// TIA Portal project "BTL2_TIA" (V17)

(* hardware
DEVICE "S7-300/ET200M station_2"  S7-300 station
   slot 0: "Rail_0"  Rail  6ES7 390-1***0-0AA0
   slot 2: "PLC_2"  CPU 314C-2 PN/DP  6ES7 314-6EH04-0AB0  V3.3
      slot 2: "PROFINET interface_1"  PN-IO
         slot 1: "Port_1"  Port
         slot 2: "Port_2"  Port
      slot 5: "DI 24/DO 16_1"  DI24/DO16
      slot 6: "AI 5/AO 2_1"  AI5/AO2
      slot 7: "Count_1"  Counter
      slot 8: "Positioning_1"  Positioning
*)

// ===== PLC "PLC_2"  CPU 314C-2 PN/DP =====

VAR_GLOBAL   // PLC tag table "I"
   "Start" AT %I0.0 : Bool;
   "Stop" AT %I0.1 : Bool;
   "Reset" AT %I0.2 : Bool;
   "Emer" AT %I0.3 : Bool;
   "Mode" AT %I0.4 : Bool;
   "S1" AT %I1.0 : Bool;   // A1
   "S2" AT %I1.1 : Bool;   // A0
   "S3" AT %I1.2 : Bool;   // B1
   "S4" AT %I1.3 : Bool;   // B0
   "S5" AT %I1.4 : Bool;   // C1
   "S6" AT %I1.5 : Bool;   // C0
   "cell" AT %I0.5 : Bool;
   "swa+" AT %I2.0 : Bool;
   "swa-" AT %I2.1 : Bool;
   "swb+" AT %I2.2 : Bool;
   "swb-" AT %I2.3 : Bool;
   "swc+" AT %I2.4 : Bool;
   "swc-" AT %I2.5 : Bool;
   "sm" AT %I2.6 : Bool;
END_VAR

VAR_GLOBAL   // PLC tag table "M"
   "k1-au" AT %M0.1 : Bool;
   "k2-au" AT %M0.2 : Bool;
   "k3-au" AT %M0.3 : Bool;
   "k4-au" AT %M0.4 : Bool;
   "k5-au" AT %M0.5 : Bool;
   "k6-au" AT %M0.6 : Bool;
   "k7-au" AT %M0.7 : Bool;
   "k0-au" AT %M0.0 : Bool;
   "cell_temp" AT %M1.0 : Bool;
   "LED_1hz" AT %M1.1 : Bool;
   "LED_Stable" AT %M1.2 : Bool;
   "au-manu" AT %M1.3 : Bool;
   "manu-au" AT %M1.4 : Bool;
   "k0-manu" AT %M1.5 : Bool;
   "protocol" AT %M1.7 : Bool;
   "k0_manu1" AT %M2.0 : Bool;
   "cell_temp_manual" AT %M2.1 : Bool;
   "stop temporary" AT %M2.2 : Bool;
   "m_err1" AT %M10.1 : Bool;
   "m_err2" AT %M10.2 : Bool;
   "m_err3" AT %M10.3 : Bool;
   "tag 1 auto" AT %M20.1 : Bool;
   "tag 2 auto" AT %M20.2 : Bool;
   "tag 1 manual" AT %M20.3 : Bool;
   "tag 2 manual" AT %M20.4 : Bool;
   "state 1" AT %M20.5 : Bool;
   "state 2" AT %M20.6 : Bool;
   "state 3" AT %M20.7 : Bool;
   "tag1" AT %M21.0 : Bool;
END_VAR

VAR_GLOBAL   // PLC tag table "Q"
   "Y1" AT %Q0.0 : Bool;   // A+
   "Y2" AT %Q0.1 : Bool;   // A-
   "Y3" AT %Q0.2 : Bool;   // B+
   "Y4" AT %Q0.3 : Bool;   // B-
   "Y5" AT %Q0.4 : Bool;   // C+
   "Y6" AT %Q0.5 : Bool;   // C-
   "M" AT %Q1.0 : Bool;
   "cell LED" AT %Q1.1 : Bool;
   "auto LED" AT %Q1.2 : Bool;
   "manual LED" AT %Q1.3 : Bool;
   "ready LED" AT %Q1.4 : Bool;
   "err1" AT %Q1.5 : Bool;
   "err2" AT %Q1.6 : Bool;
   "err3" AT %Q1.7 : Bool;
END_VAR

FUNCTION "auto" : Void   // FC1, LAD
{ S7_Optimized_Access := 'FALSE' }
VERSION : 0.1
BEGIN

REGION Network 1
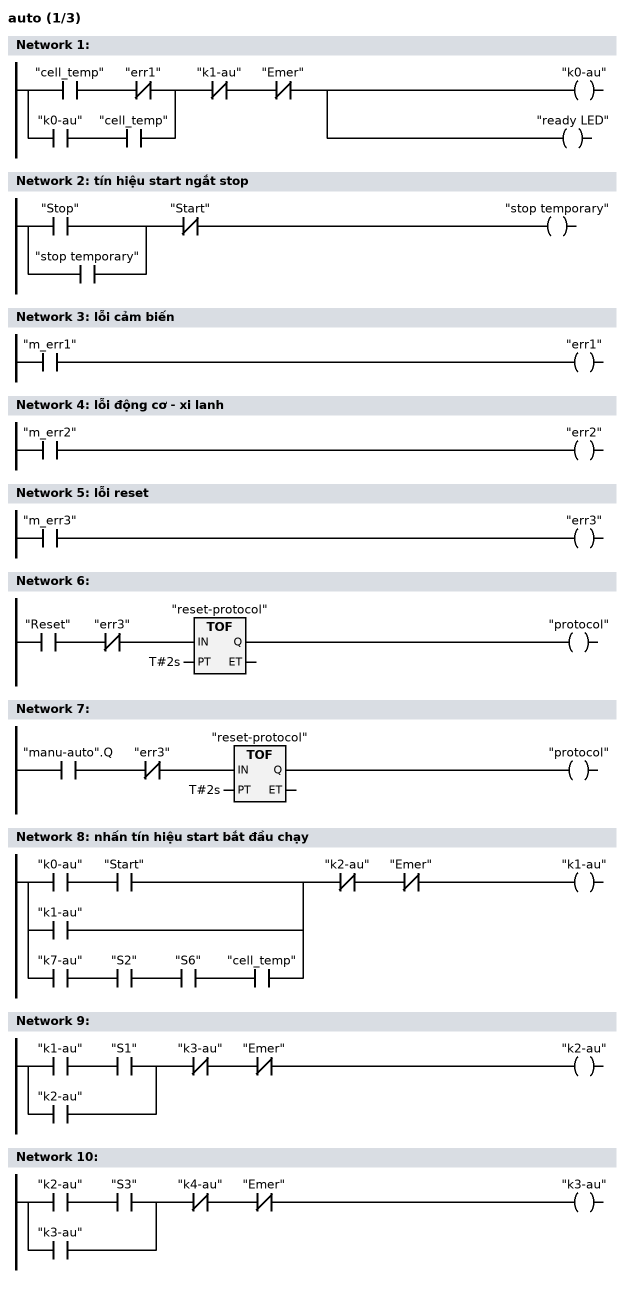
   RUNG wire#powerrail
      Contact( "cell_temp" )
      I_Contact( "err1" )
      wire#w1
      I_Contact( "k1-au" )
      I_Contact( "Emer" )
      wire#w2
      Coil( "k0-au" )
   END_RUNG
   RUNG wire#powerrail
      Contact( "k0-au" )
      Contact( "cell_temp" )
   END_RUNG wire#w1
   RUNG wire#w2
      Coil( "ready LED" )
   END_RUNG
   // the same network as SCL:
   "k0-au" := (("cell_temp" AND NOT "err1") OR ("k0-au" AND "cell_temp")) AND NOT "k1-au" AND NOT "Emer";
   "ready LED" := "k0-au";
END_REGION

REGION Network 2: tín hiệu start ngắt stop
   RUNG wire#powerrail
      Contact( "Stop" )
      wire#w1
      I_Contact( "Start" )
      Coil( "stop temporary" )
   END_RUNG
   RUNG wire#powerrail
      Contact( "stop temporary" )
   END_RUNG wire#w1
   // the same network as SCL:
   "stop temporary" := ("Stop" OR "stop temporary") AND NOT "Start";
END_REGION

REGION Network 3: lỗi cảm biến
   RUNG wire#powerrail
      Contact( "m_err1" )
      Coil( "err1" )
   END_RUNG
   // the same network as SCL:
   "err1" := "m_err1";
END_REGION

REGION Network 4: lỗi động cơ - xi lanh
   RUNG wire#powerrail
      Contact( "m_err2" )
      Coil( "err2" )
   END_RUNG
   // the same network as SCL:
   "err2" := "m_err2";
END_REGION

REGION Network 5: lỗi reset
   RUNG wire#powerrail
      Contact( "m_err3" )
      Coil( "err3" )
   END_RUNG
   // the same network as SCL:
   "err3" := "m_err3";
END_REGION

REGION Network 6
   "reset-protocol".TOF(IN := "Reset" AND NOT "err3", PT := T#2s);
   "protocol" := "reset-protocol".Q;
END_REGION

REGION Network 7
   "reset-protocol".TOF(IN := "manu-auto".Q AND NOT "err3", PT := T#2s);
   "protocol" := "reset-protocol".Q;
END_REGION

REGION Network 8: nhấn tín hiệu start bắt đầu chạy
   RUNG wire#powerrail
      Contact( "k0-au" )
      Contact( "Start" )
      wire#w1
      I_Contact( "k2-au" )
      I_Contact( "Emer" )
      Coil( "k1-au" )
   END_RUNG
   RUNG wire#powerrail
      Contact( "k1-au" )
   END_RUNG wire#w1
   RUNG wire#powerrail
      Contact( "k7-au" )
      Contact( "S2" )
      Contact( "S6" )
      Contact( "cell_temp" )
   END_RUNG wire#w1
   // the same network as SCL:
   "k1-au" := (("k0-au" AND "Start") OR "k1-au" OR ("k7-au" AND "S2" AND "S6" AND "cell_temp")) AND NOT "k2-au" AND NOT "Emer";
END_REGION

REGION Network 9
   RUNG wire#powerrail
      Contact( "k1-au" )
      Contact( "S1" )
      wire#w1
      I_Contact( "k3-au" )
      I_Contact( "Emer" )
      Coil( "k2-au" )
   END_RUNG
   RUNG wire#powerrail
      Contact( "k2-au" )
   END_RUNG wire#w1
   // the same network as SCL:
   "k2-au" := (("k1-au" AND "S1") OR "k2-au") AND NOT "k3-au" AND NOT "Emer";
END_REGION

REGION Network 10
   RUNG wire#powerrail
      Contact( "k2-au" )
      Contact( "S3" )
      wire#w1
      I_Contact( "k4-au" )
      I_Contact( "Emer" )
      Coil( "k3-au" )
   END_RUNG
   RUNG wire#powerrail
      Contact( "k3-au" )
   END_RUNG wire#w1
   // the same network as SCL:
   "k3-au" := (("k2-au" AND "S3") OR "k3-au") AND NOT "k4-au" AND NOT "Emer";
END_REGION

REGION Network 11
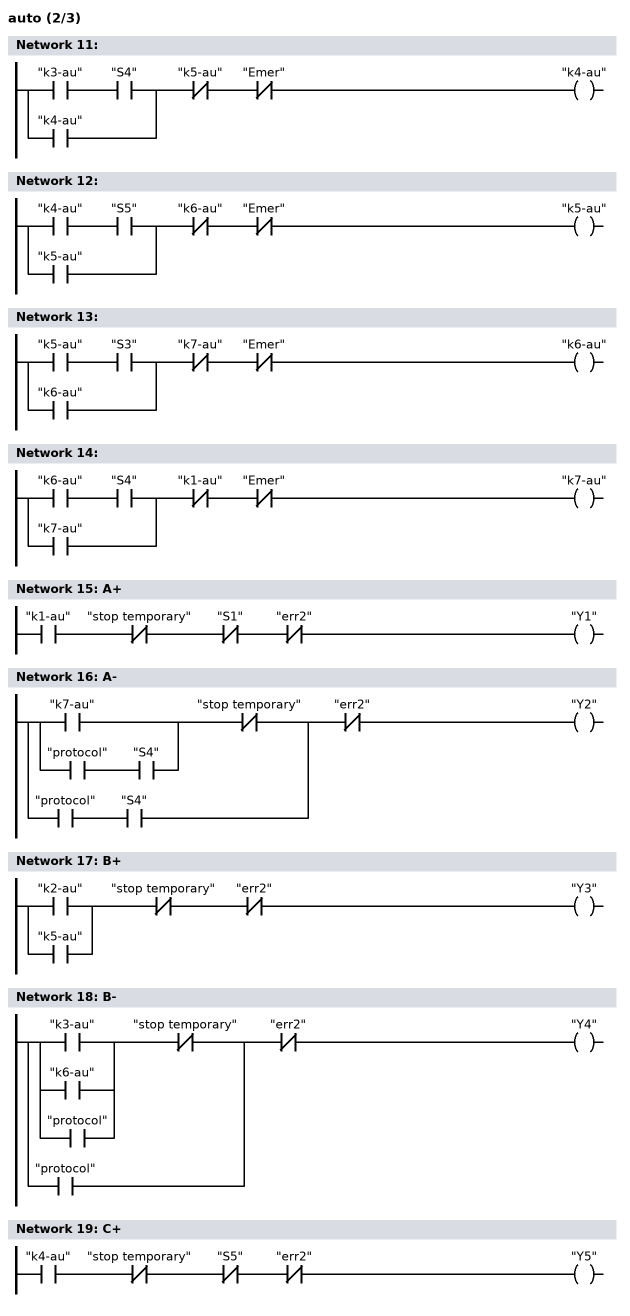
   RUNG wire#powerrail
      Contact( "k3-au" )
      Contact( "S4" )
      wire#w1
      I_Contact( "k5-au" )
      I_Contact( "Emer" )
      Coil( "k4-au" )
   END_RUNG
   RUNG wire#powerrail
      Contact( "k4-au" )
   END_RUNG wire#w1
   // the same network as SCL:
   "k4-au" := (("k3-au" AND "S4") OR "k4-au") AND NOT "k5-au" AND NOT "Emer";
END_REGION

REGION Network 12
   RUNG wire#powerrail
      Contact( "k4-au" )
      Contact( "S5" )
      wire#w1
      I_Contact( "k6-au" )
      I_Contact( "Emer" )
      Coil( "k5-au" )
   END_RUNG
   RUNG wire#powerrail
      Contact( "k5-au" )
   END_RUNG wire#w1
   // the same network as SCL:
   "k5-au" := (("k4-au" AND "S5") OR "k5-au") AND NOT "k6-au" AND NOT "Emer";
END_REGION

REGION Network 13
   RUNG wire#powerrail
      Contact( "k5-au" )
      Contact( "S3" )
      wire#w1
      I_Contact( "k7-au" )
      I_Contact( "Emer" )
      Coil( "k6-au" )
   END_RUNG
   RUNG wire#powerrail
      Contact( "k6-au" )
   END_RUNG wire#w1
   // the same network as SCL:
   "k6-au" := (("k5-au" AND "S3") OR "k6-au") AND NOT "k7-au" AND NOT "Emer";
END_REGION

REGION Network 14
   RUNG wire#powerrail
      Contact( "k6-au" )
      Contact( "S4" )
      wire#w1
      I_Contact( "k1-au" )
      I_Contact( "Emer" )
      Coil( "k7-au" )
   END_RUNG
   RUNG wire#powerrail
      Contact( "k7-au" )
   END_RUNG wire#w1
   // the same network as SCL:
   "k7-au" := (("k6-au" AND "S4") OR "k7-au") AND NOT "k1-au" AND NOT "Emer";
END_REGION

REGION Network 15: A+
   RUNG wire#powerrail
      Contact( "k1-au" )
      I_Contact( "stop temporary" )
      I_Contact( "S1" )
      I_Contact( "err2" )
      Coil( "Y1" )
   END_RUNG
   // the same network as SCL:
   "Y1" := "k1-au" AND NOT "stop temporary" AND NOT "S1" AND NOT "err2";
END_REGION

REGION Network 16: A-
   RUNG wire#powerrail
      Contact( "k7-au" )
      wire#w1
      I_Contact( "stop temporary" )
      wire#w2
      I_Contact( "err2" )
      Coil( "Y2" )
   END_RUNG
   RUNG wire#powerrail
      Contact( "protocol" )
      Contact( "S4" )
   END_RUNG wire#w1
   RUNG wire#powerrail
      Contact( "protocol" )
      Contact( "S4" )
   END_RUNG wire#w2
   // the same network as SCL:
   "Y2" := ((("k7-au" OR ("protocol" AND "S4")) AND NOT "stop temporary") OR ("protocol" AND "S4")) AND NOT "err2";
END_REGION

REGION Network 17: B+
   RUNG wire#powerrail
      Contact( "k2-au" )
      wire#w1
      I_Contact( "stop temporary" )
      I_Contact( "err2" )
      Coil( "Y3" )
   END_RUNG
   RUNG wire#powerrail
      Contact( "k5-au" )
   END_RUNG wire#w1
   // the same network as SCL:
   "Y3" := ("k2-au" OR "k5-au") AND NOT "stop temporary" AND NOT "err2";
END_REGION

REGION Network 18: B-
   RUNG wire#powerrail
      Contact( "k3-au" )
      wire#w1
      I_Contact( "stop temporary" )
      wire#w2
      I_Contact( "err2" )
      Coil( "Y4" )
   END_RUNG
   RUNG wire#powerrail
      Contact( "k6-au" )
   END_RUNG wire#w1
   RUNG wire#powerrail
      Contact( "protocol" )
   END_RUNG wire#w1
   RUNG wire#powerrail
      Contact( "protocol" )
   END_RUNG wire#w2
   // the same network as SCL:
   "Y4" := ((("k3-au" OR "k6-au" OR "protocol") AND NOT "stop temporary") OR "protocol") AND NOT "err2";
END_REGION

REGION Network 19: C+
   RUNG wire#powerrail
      Contact( "k4-au" )
      I_Contact( "stop temporary" )
      I_Contact( "S5" )
      I_Contact( "err2" )
      Coil( "Y5" )
   END_RUNG
   // the same network as SCL:
   "Y5" := "k4-au" AND NOT "stop temporary" AND NOT "S5" AND NOT "err2";
END_REGION

REGION Network 20: C-
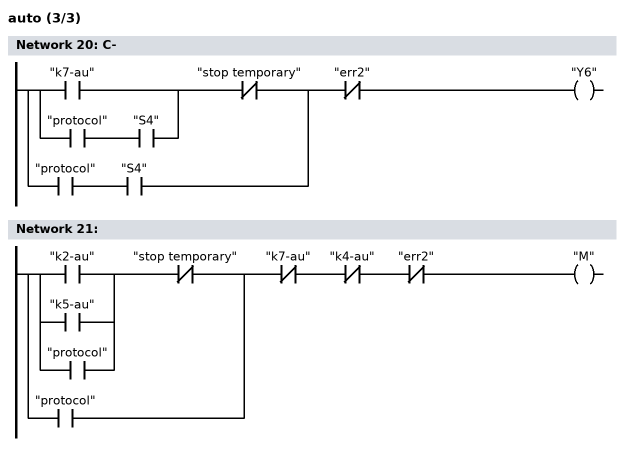
   RUNG wire#powerrail
      Contact( "k7-au" )
      wire#w1
      I_Contact( "stop temporary" )
      wire#w2
      I_Contact( "err2" )
      Coil( "Y6" )
   END_RUNG
   RUNG wire#powerrail
      Contact( "protocol" )
      Contact( "S4" )
   END_RUNG wire#w1
   RUNG wire#powerrail
      Contact( "protocol" )
      Contact( "S4" )
   END_RUNG wire#w2
   // the same network as SCL:
   "Y6" := ((("k7-au" OR ("protocol" AND "S4")) AND NOT "stop temporary") OR ("protocol" AND "S4")) AND NOT "err2";
END_REGION

REGION Network 21
   RUNG wire#powerrail
      Contact( "k2-au" )
      wire#w1
      I_Contact( "stop temporary" )
      wire#w2
      I_Contact( "k7-au" )
      I_Contact( "k4-au" )
      I_Contact( "err2" )
      Coil( "M" )
   END_RUNG
   RUNG wire#powerrail
      Contact( "k5-au" )
   END_RUNG wire#w1
   RUNG wire#powerrail
      Contact( "protocol" )
   END_RUNG wire#w1
   RUNG wire#powerrail
      Contact( "protocol" )
   END_RUNG wire#w2
   // the same network as SCL:
   "M" := ((("k2-au" OR "k5-au" OR "protocol") AND NOT "stop temporary") OR "protocol") AND NOT "k7-au" AND NOT "k4-au" AND NOT "err2";
END_REGION
END_FUNCTION

FUNCTION "manu" : Void   // FC2, LAD
{ S7_Optimized_Access := 'FALSE' }
VERSION : 0.1
   VAR_TEMP   // added for the SCL form of the ladder/FBD networks
      _w1 : Bool;
      _w2 : Bool;
   END_VAR
BEGIN

REGION Network 1: reset-from-auto
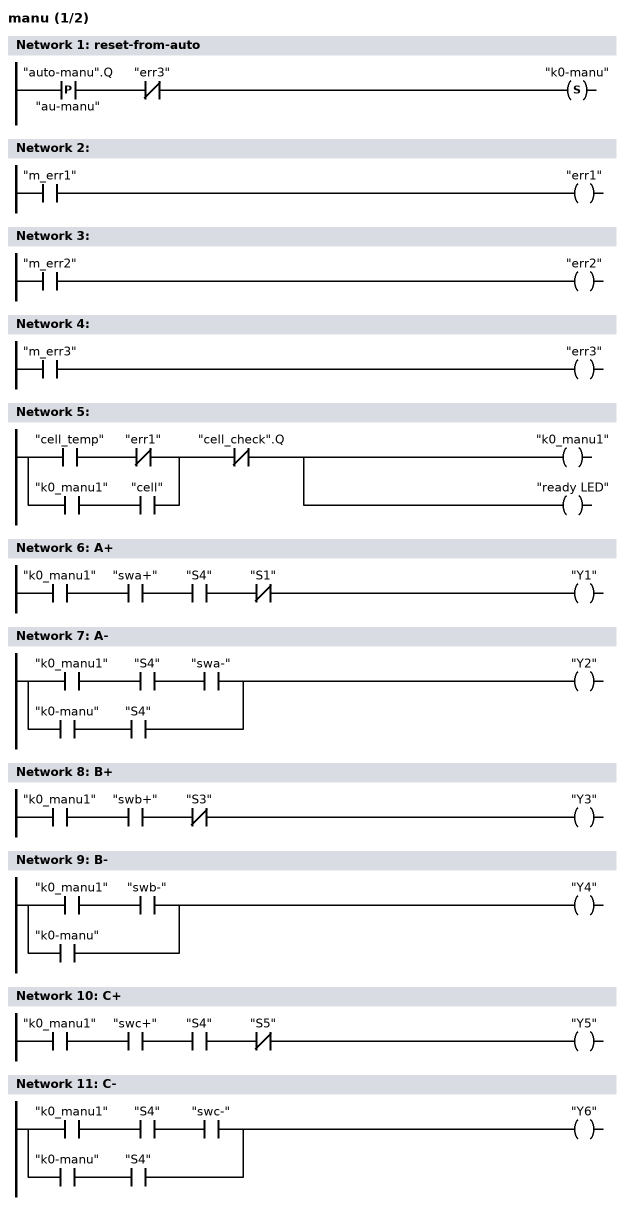
   RUNG wire#powerrail
      P_Contact(operand := "auto-manu".Q, bit := "au-manu")
      I_Contact( "err3" )
      S_Coil( "k0-manu" )
   END_RUNG
   // the same network as SCL:
   #_w1 := "auto-manu".Q AND NOT "au-manu";   // rising edge of "auto-manu".Q
   "au-manu" := "auto-manu".Q;
   IF #_w1 AND NOT "err3" THEN "k0-manu" := TRUE; END_IF;
END_REGION

REGION Network 2
   RUNG wire#powerrail
      Contact( "m_err1" )
      Coil( "err1" )
   END_RUNG
   // the same network as SCL:
   "err1" := "m_err1";
END_REGION

REGION Network 3
   RUNG wire#powerrail
      Contact( "m_err2" )
      Coil( "err2" )
   END_RUNG
   // the same network as SCL:
   "err2" := "m_err2";
END_REGION

REGION Network 4
   RUNG wire#powerrail
      Contact( "m_err3" )
      Coil( "err3" )
   END_RUNG
   // the same network as SCL:
   "err3" := "m_err3";
END_REGION

REGION Network 5
   RUNG wire#powerrail
      Contact( "cell_temp" )
      I_Contact( "err1" )
      wire#w1
      I_Contact( "cell_check".Q )
      wire#w2
      Coil( "k0_manu1" )
   END_RUNG
   RUNG wire#powerrail
      Contact( "k0_manu1" )
      Contact( "cell" )
   END_RUNG wire#w1
   RUNG wire#w2
      Coil( "ready LED" )
   END_RUNG
   // the same network as SCL:
   "k0_manu1" := (("cell_temp" AND NOT "err1") OR ("k0_manu1" AND "cell")) AND NOT "cell_check".Q;
   "ready LED" := "k0_manu1";
END_REGION

REGION Network 6: A+
   RUNG wire#powerrail
      Contact( "k0_manu1" )
      Contact( "swa+" )
      Contact( "S4" )
      I_Contact( "S1" )
      Coil( "Y1" )
   END_RUNG
   // the same network as SCL:
   "Y1" := "k0_manu1" AND "swa+" AND "S4" AND NOT "S1";
END_REGION

REGION Network 7: A-
   RUNG wire#powerrail
      Contact( "k0_manu1" )
      Contact( "S4" )
      Contact( "swa-" )
      wire#w1
      Coil( "Y2" )
   END_RUNG
   RUNG wire#powerrail
      Contact( "k0-manu" )
      Contact( "S4" )
   END_RUNG wire#w1
   // the same network as SCL:
   "Y2" := ("k0_manu1" AND "S4" AND "swa-") OR ("k0-manu" AND "S4");
END_REGION

REGION Network 8: B+
   RUNG wire#powerrail
      Contact( "k0_manu1" )
      Contact( "swb+" )
      I_Contact( "S3" )
      Coil( "Y3" )
   END_RUNG
   // the same network as SCL:
   "Y3" := "k0_manu1" AND "swb+" AND NOT "S3";
END_REGION

REGION Network 9: B-
   RUNG wire#powerrail
      Contact( "k0_manu1" )
      Contact( "swb-" )
      wire#w1
      Coil( "Y4" )
   END_RUNG
   RUNG wire#powerrail
      Contact( "k0-manu" )
   END_RUNG wire#w1
   // the same network as SCL:
   "Y4" := ("k0_manu1" AND "swb-") OR "k0-manu";
END_REGION

REGION Network 10: C+
   RUNG wire#powerrail
      Contact( "k0_manu1" )
      Contact( "swc+" )
      Contact( "S4" )
      I_Contact( "S5" )
      Coil( "Y5" )
   END_RUNG
   // the same network as SCL:
   "Y5" := "k0_manu1" AND "swc+" AND "S4" AND NOT "S5";
END_REGION

REGION Network 11: C-
   RUNG wire#powerrail
      Contact( "k0_manu1" )
      Contact( "S4" )
      Contact( "swc-" )
      wire#w1
      Coil( "Y6" )
   END_RUNG
   RUNG wire#powerrail
      Contact( "k0-manu" )
      Contact( "S4" )
   END_RUNG wire#w1
   // the same network as SCL:
   "Y6" := ("k0_manu1" AND "S4" AND "swc-") OR ("k0-manu" AND "S4");
END_REGION

REGION Network 12
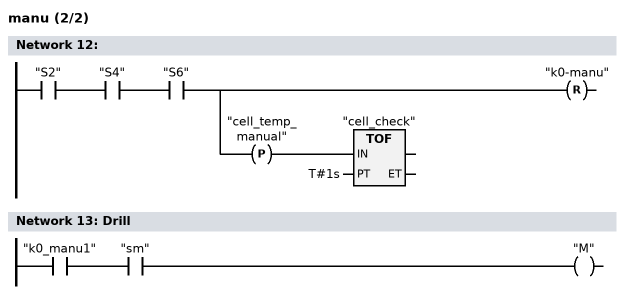
   #_w1 := "S2" AND "S4" AND "S6";
   IF #_w1 THEN "k0-manu" := FALSE; END_IF;
   #_w2 := #_w1 AND NOT "cell_temp_manual";   // rising edge
   "cell_temp_manual" := #_w1;
   "cell_check".TOF(IN := #_w2, PT := T#1s);
END_REGION

REGION Network 13: Drill
   RUNG wire#powerrail
      Contact( "k0_manu1" )
      Contact( "sm" )
      Coil( "M" )
   END_RUNG
   // the same network as SCL:
   "M" := "k0_manu1" AND "sm";
END_REGION
END_FUNCTION

FUNCTION "cell_blink_auto" : Void   // FC3, LAD
{ S7_Optimized_Access := 'FALSE' }
VERSION : 0.1
   VAR_TEMP   // added for the SCL form of the ladder/FBD networks
      _w1 : Bool;
      _w2 : Bool;
      _w3 : Bool;
   END_VAR
BEGIN

REGION Network 1
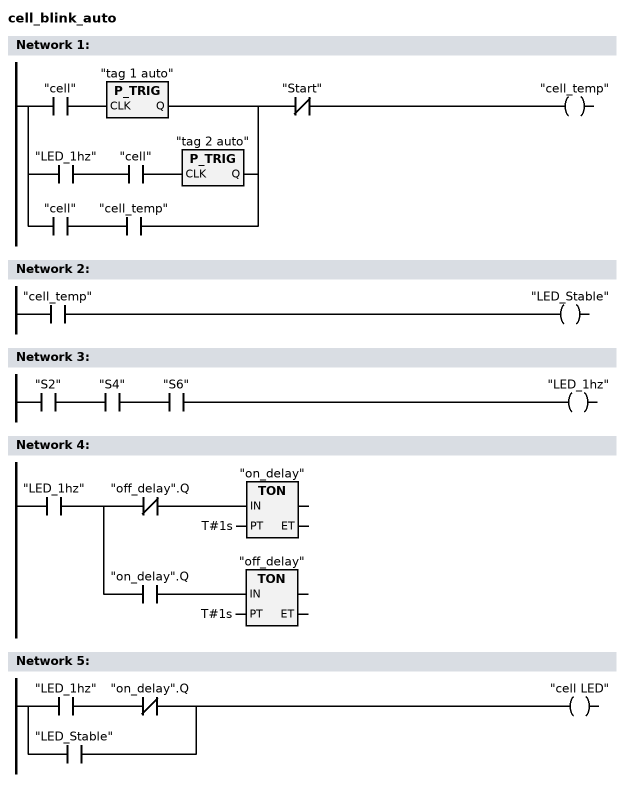
   RUNG wire#powerrail
      Contact( "cell" )
      P_Trig( "tag 1 auto" )
      wire#w1
      I_Contact( "Start" )
      Coil( "cell_temp" )
   END_RUNG
   RUNG wire#powerrail
      Contact( "LED_1hz" )
      Contact( "cell" )
      P_Trig( "tag 2 auto" )
   END_RUNG wire#w1
   RUNG wire#powerrail
      Contact( "cell" )
      Contact( "cell_temp" )
   END_RUNG wire#w1
   // the same network as SCL:
   #_w1 := "cell" AND NOT "tag 1 auto";   // rising edge
   "tag 1 auto" := "cell";
   #_w2 := "LED_1hz" AND "cell";
   #_w3 := #_w2 AND NOT "tag 2 auto";   // rising edge
   "tag 2 auto" := #_w2;
   "cell_temp" := (#_w1 OR #_w3 OR ("cell" AND "cell_temp")) AND NOT "Start";
END_REGION

REGION Network 2
   RUNG wire#powerrail
      Contact( "cell_temp" )
      Coil( "LED_Stable" )
   END_RUNG
   // the same network as SCL:
   "LED_Stable" := "cell_temp";
END_REGION

REGION Network 3
   RUNG wire#powerrail
      Contact( "S2" )
      Contact( "S4" )
      Contact( "S6" )
      Coil( "LED_1hz" )
   END_RUNG
   // the same network as SCL:
   "LED_1hz" := "S2" AND "S4" AND "S6";
END_REGION

REGION Network 4
   "on_delay".TON(IN := "LED_1hz" AND NOT "off_delay".Q, PT := T#1s);
   "off_delay".TON(IN := "LED_1hz" AND "on_delay".Q, PT := T#1s);
END_REGION

REGION Network 5
   RUNG wire#powerrail
      Contact( "LED_1hz" )
      I_Contact( "on_delay".Q )
      wire#w1
      Coil( "cell LED" )
   END_RUNG
   RUNG wire#powerrail
      Contact( "LED_Stable" )
   END_RUNG wire#w1
   // the same network as SCL:
   "cell LED" := ("LED_1hz" AND NOT "on_delay".Q) OR "LED_Stable";
END_REGION
END_FUNCTION

FUNCTION "cell_blink_manu" : Void   // FC4, LAD
{ S7_Optimized_Access := 'FALSE' }
VERSION : 0.1
BEGIN

REGION Network 1
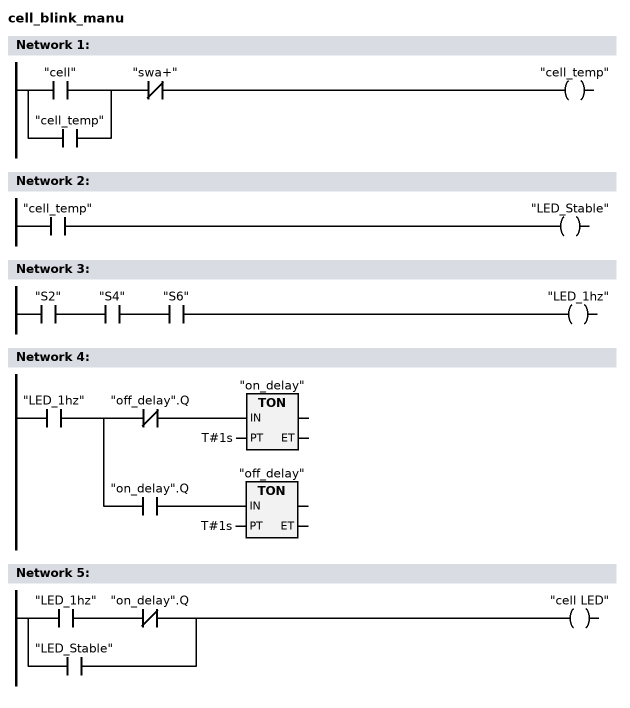
   RUNG wire#powerrail
      Contact( "cell" )
      wire#w1
      I_Contact( "swa+" )
      Coil( "cell_temp" )
   END_RUNG
   RUNG wire#powerrail
      Contact( "cell_temp" )
   END_RUNG wire#w1
   // the same network as SCL:
   "cell_temp" := ("cell" OR "cell_temp") AND NOT "swa+";
END_REGION

REGION Network 2
   RUNG wire#powerrail
      Contact( "cell_temp" )
      Coil( "LED_Stable" )
   END_RUNG
   // the same network as SCL:
   "LED_Stable" := "cell_temp";
END_REGION

REGION Network 3
   RUNG wire#powerrail
      Contact( "S2" )
      Contact( "S4" )
      Contact( "S6" )
      Coil( "LED_1hz" )
   END_RUNG
   // the same network as SCL:
   "LED_1hz" := "S2" AND "S4" AND "S6";
END_REGION

REGION Network 4
   "on_delay".TON(IN := "LED_1hz" AND NOT "off_delay".Q, PT := T#1s);
   "off_delay".TON(IN := "LED_1hz" AND "on_delay".Q, PT := T#1s);
END_REGION

REGION Network 5
   RUNG wire#powerrail
      Contact( "LED_1hz" )
      I_Contact( "on_delay".Q )
      wire#w1
      Coil( "cell LED" )
   END_RUNG
   RUNG wire#powerrail
      Contact( "LED_Stable" )
   END_RUNG wire#w1
   // the same network as SCL:
   "cell LED" := ("LED_1hz" AND NOT "on_delay".Q) OR "LED_Stable";
END_REGION
END_FUNCTION

ORGANIZATION_BLOCK "Main"   // OB1, LAD
TITLE = "Main Program Sweep (Cycle)"
{ S7_Optimized_Access := 'FALSE' }
VERSION : 0.1
   VAR_TEMP
      OB1_EV_CLASS : Byte;   // Bits 0-3 = 1 (Coming event), Bits 4-7 = 1 (Event class 1)
      OB1_SCAN_1 : Byte;   // 1 (Cold restart scan 1 of OB 1), 3 (Scan 2-n of OB 1)
      OB1_PRIORITY : Byte;   // Priority of OB Execution
      OB1_OB_NUMBR : Byte;   // 1 (Organization block 1, OB1)
      OB1_RESERVED_1 : Byte;   // Reserved for system
      OB1_RESERVED_2 : Byte;   // Reserved for system
      OB1_PREV_CYCLE : Int;   // Cycle time of previous OB1 scan (milliseconds)
      OB1_MIN_CYCLE : Int;   // Minimum cycle time of OB1 (milliseconds)
      OB1_MAX_CYCLE : Int;   // Maximum cycle time of OB1 (milliseconds)
      OB1_DATE_TIME : Date_And_Time;   // Date and time OB1 started
   END_VAR
   VAR_TEMP   // added for the SCL form of the ladder/FBD networks
      _w1 : Bool;
      _w2 : Bool;
   END_VAR
BEGIN

REGION Network 1: auto mode
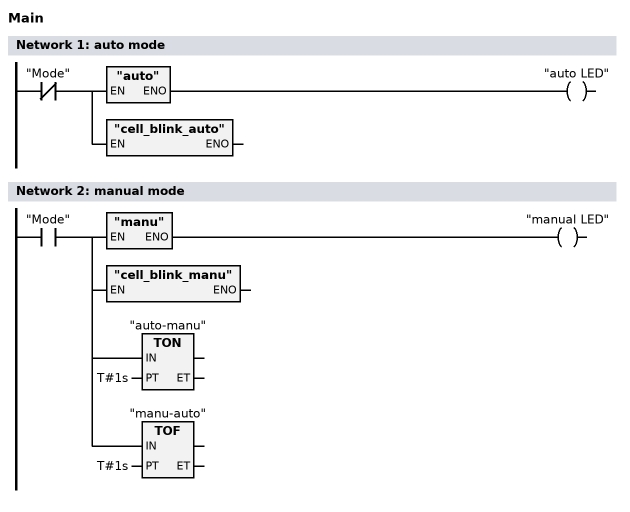
   RUNG wire#powerrail
      I_Contact( "Mode" )
      wire#w1
      "auto"()
      Coil( "auto LED" )
   END_RUNG
   RUNG wire#w1
      "cell_blink_auto"()
   END_RUNG
   // the same network as SCL:
   #_w2 := NOT "Mode";
   "auto"(EN := NOT "Mode", ENO => #_w1);
   "auto LED" := #_w1;
   IF #_w2 THEN "cell_blink_auto"(); END_IF;
END_REGION

REGION Network 2: manual mode
   #_w2 := "Mode";
   "manu"(EN := "Mode", ENO => #_w1);
   "manual LED" := #_w1;
   IF #_w2 THEN "cell_blink_manu"(); END_IF;
   "auto-manu".TON(IN := #_w2, PT := T#1s);
   "manu-auto".TOF(IN := #_w2, PT := T#1s);
END_REGION
END_ORGANIZATION_BLOCK